PROGRAM MAIN
VAR
END_VAR

END_PROGRAM

(* stored: Version 1.1.0.1
   POU MAIN: Id {567ebe3e-ff42-438b-8194-78ca79d14516} *)
